// TwinCAT 3 PLC project PlcTemplate
// Title: PlcTemplate
// Company: Vortex.Library
// ProjectVersion: 0.0.0.0
// ProgramVersion: 3.1.4023.0
// libraries:
//   Tc2_Standard, * (Beckhoff Automation GmbH)
//   Tc2_System, * (Beckhoff Automation GmbH)
//   Tc3_Module, * (Beckhoff Automation GmbH)
// project tree:
//   / PlcTask.TcTTO (not stored)
//   POUs/ fbSampleComponent.TcPOU (not stored), MAIN.TcPOU
// real-time tasks:
//   TASK PlcTask: cycle T#10ms, priority 20, ADS port 350

// ---- POUs/MAIN.TcPOU
PROGRAM MAIN
VAR
	_unitTestExample : fbSampleComponent;
END_VAR

_unitTestExample.Cyclic();

END_PROGRAM
